PROGRAM SPIDER_DEMO
VAR
	SPIDER_ACCESS: SPIDER_ACCESS;
	IP_CONTROL: IP_CONTROL;
	S_BUF: NETWORK_BUFFER;
	R_BUF: NETWORK_BUFFER;
	MODE: BYTE := 1;
	IP_C: IP_C;
	VALUE: STRING;
	VAR_NAME: STRING(40) := 'RTC_SECONDS';
	ERROR: DWORD;
END_VAR
VAR // added by the converter: edge detectors and wires of the graphical bodies
    _w1 : ANY;
END_VAR

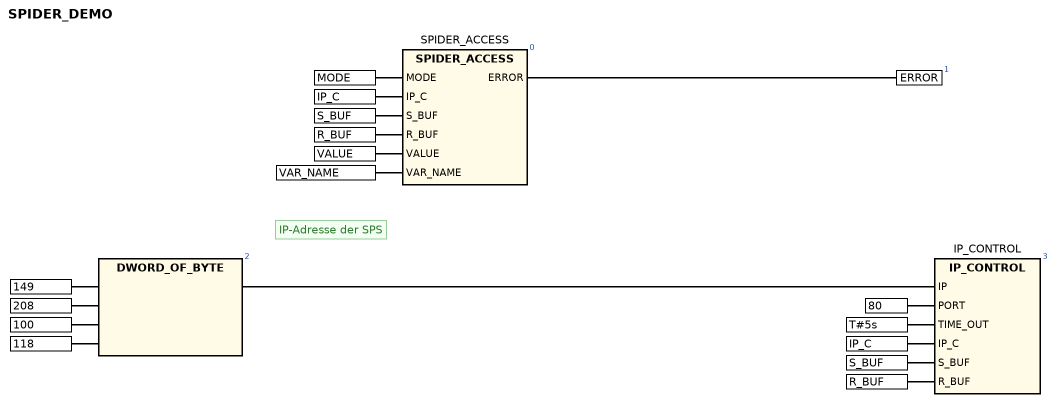
SPIDER_ACCESS(
    MODE := MODE,
    IP_C := IP_C,
    S_BUF := S_BUF,
    R_BUF := R_BUF,
    VALUE := VALUE,
    VAR_NAME := VAR_NAME);
ERROR := SPIDER_ACCESS.ERROR;
// IP-Adresse der SPS
_w1 := DWORD_OF_BYTE(149, 208, 100, 118);
IP_CONTROL(IP := _w1, PORT := 80, TIME_OUT := T#5s, IP_C := IP_C, S_BUF := S_BUF, R_BUF := R_BUF);

END_PROGRAM

(* stored: Version 1.1.0.1, ProductVersion 3.1.4024.9
   POU SPIDER_DEMO: Id {0438ae26-ca8a-4217-abda-89c8058bddcc}, SpecialFunc None *)
